PROGRAM pouStation2
VAR
	stationMode: FB_Mode;
	tCalcNumberOfPages: REAL;
	ceil: REAL;
	PartBuild: FB_PartBuild;
	retvall: UDINT;
	// TODO
	tPartPresent: BOOL;
	stationPower: FB_PowerDelay;
	
	task1: FB_Task;
	task2: FB_Task;
	task3: FB_Task;
	task4: FB_Task;
	task5: FB_Task;
	task6: FB_Task;
	task7: FB_Task;
	task8: FB_Task;
	task9: FB_Task;
	task10: FB_Task;
	task11: FB_Task;
	task12: FB_Task;
	task13: FB_Task;
	task14: FB_Task;
	task15: FB_Task;
	task16: FB_Task;
	task17: FB_Task;
	task18: FB_Task;
	task19: FB_Task;
	task20: FB_Task;
	checkTasks: FB_CheckTasks;
END_VAR

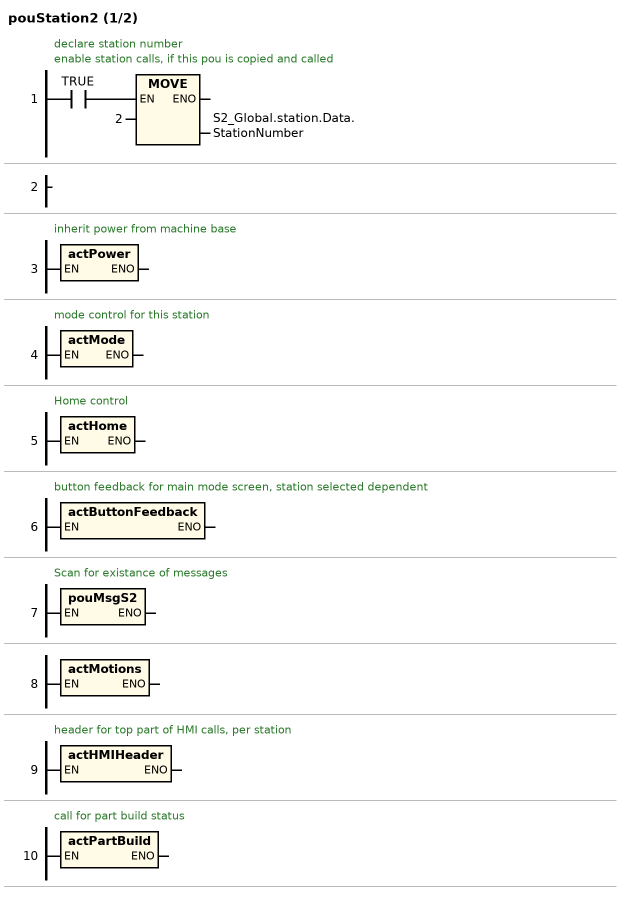
// NETWORK 1
// declare station number
// enable station calls, if this pou is copied and called
S2_Global.station.Data.StationNumber := 2;

// NETWORK 2

// NETWORK 3
// inherit power from machine base
actPower();

// NETWORK 4
// mode control for this station
actMode();

// NETWORK 5
// Home control
actHome();

// NETWORK 6
// button feedback for main mode screen, station selected dependent
actButtonFeedback();

// NETWORK 7
// Scan for existance of messages
pouMsgS2();

// NETWORK 8
actMotions();

// NETWORK 9
// header for top part of HMI calls, per station
actHMIHeader();

// NETWORK 10
// call for part build status
actPartBuild();

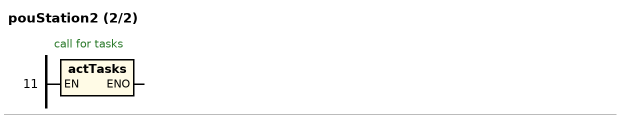
// NETWORK 11
// call for tasks
actTasks();

ACTION actButtonFeedback:
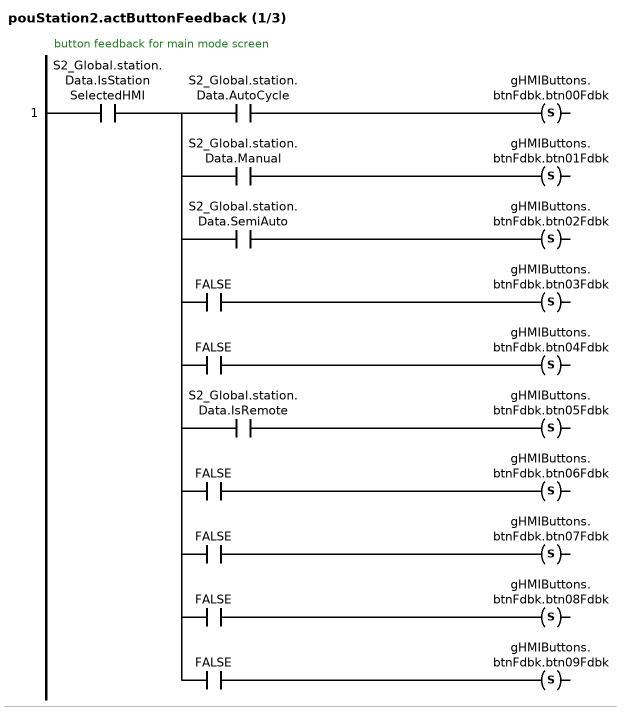
// NETWORK 1
// button feedback for main mode screen
gHMIButtons.btnFdbk.btn00Fdbk S= S2_Global.station.Data.IsStationSelectedHMI AND S2_Global.station.Data.AutoCycle;
gHMIButtons.btnFdbk.btn01Fdbk S= S2_Global.station.Data.IsStationSelectedHMI AND S2_Global.station.Data.Manual;
gHMIButtons.btnFdbk.btn02Fdbk S= S2_Global.station.Data.IsStationSelectedHMI AND S2_Global.station.Data.SemiAuto;
gHMIButtons.btnFdbk.btn03Fdbk S= S2_Global.station.Data.IsStationSelectedHMI AND FALSE;
gHMIButtons.btnFdbk.btn04Fdbk S= S2_Global.station.Data.IsStationSelectedHMI AND FALSE;
gHMIButtons.btnFdbk.btn05Fdbk S= S2_Global.station.Data.IsStationSelectedHMI AND S2_Global.station.Data.IsRemote;
gHMIButtons.btnFdbk.btn06Fdbk S= S2_Global.station.Data.IsStationSelectedHMI AND FALSE;
gHMIButtons.btnFdbk.btn07Fdbk S= S2_Global.station.Data.IsStationSelectedHMI AND FALSE;
gHMIButtons.btnFdbk.btn08Fdbk S= S2_Global.station.Data.IsStationSelectedHMI AND FALSE;
gHMIButtons.btnFdbk.btn09Fdbk S= S2_Global.station.Data.IsStationSelectedHMI AND FALSE;

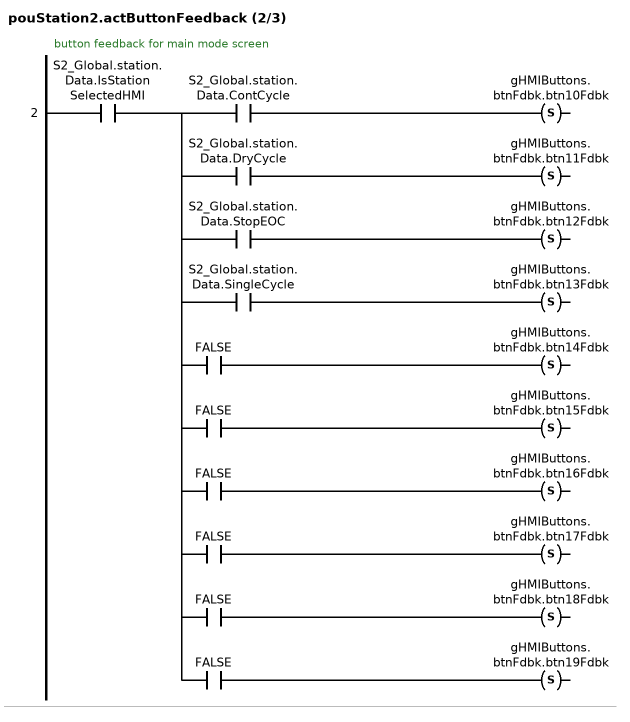
// NETWORK 2
// button feedback for main mode screen
gHMIButtons.btnFdbk.btn10Fdbk S= S2_Global.station.Data.IsStationSelectedHMI AND S2_Global.station.Data.ContCycle;
gHMIButtons.btnFdbk.btn11Fdbk S= S2_Global.station.Data.IsStationSelectedHMI AND S2_Global.station.Data.DryCycle;
gHMIButtons.btnFdbk.btn12Fdbk S= S2_Global.station.Data.IsStationSelectedHMI AND S2_Global.station.Data.StopEOC;
gHMIButtons.btnFdbk.btn13Fdbk S= S2_Global.station.Data.IsStationSelectedHMI AND S2_Global.station.Data.SingleCycle;
gHMIButtons.btnFdbk.btn14Fdbk S= S2_Global.station.Data.IsStationSelectedHMI AND FALSE;
gHMIButtons.btnFdbk.btn15Fdbk S= S2_Global.station.Data.IsStationSelectedHMI AND FALSE;
gHMIButtons.btnFdbk.btn16Fdbk S= S2_Global.station.Data.IsStationSelectedHMI AND FALSE;
gHMIButtons.btnFdbk.btn17Fdbk S= S2_Global.station.Data.IsStationSelectedHMI AND FALSE;
gHMIButtons.btnFdbk.btn18Fdbk S= S2_Global.station.Data.IsStationSelectedHMI AND FALSE;
gHMIButtons.btnFdbk.btn19Fdbk S= S2_Global.station.Data.IsStationSelectedHMI AND FALSE;

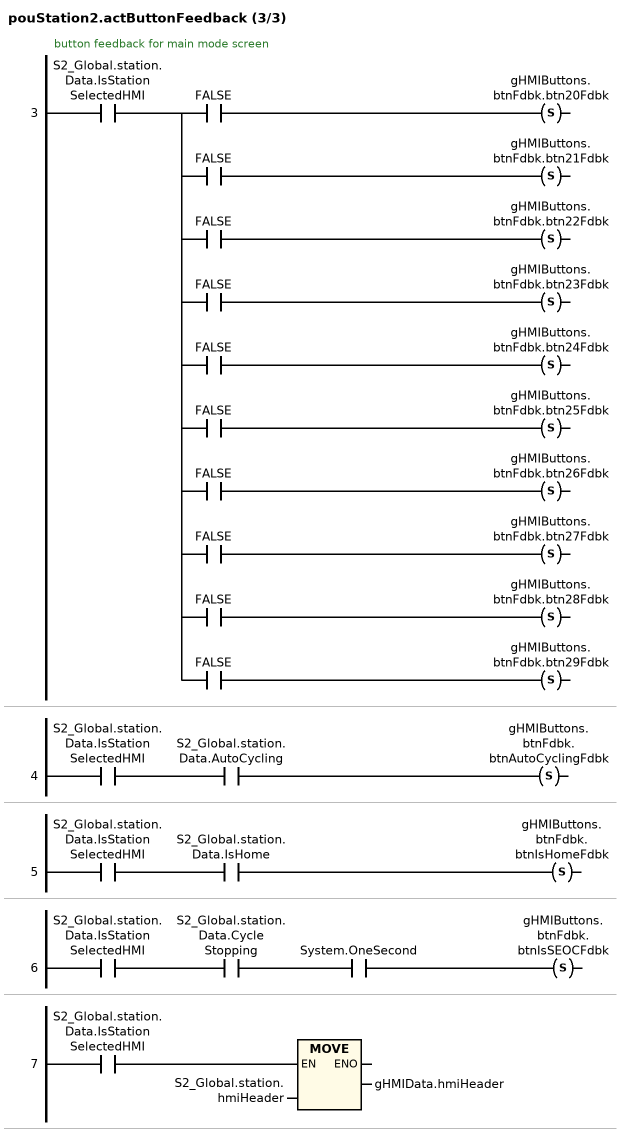
// NETWORK 3
// button feedback for main mode screen
gHMIButtons.btnFdbk.btn20Fdbk S= S2_Global.station.Data.IsStationSelectedHMI AND FALSE;
gHMIButtons.btnFdbk.btn21Fdbk S= S2_Global.station.Data.IsStationSelectedHMI AND FALSE;
gHMIButtons.btnFdbk.btn22Fdbk S= S2_Global.station.Data.IsStationSelectedHMI AND FALSE;
gHMIButtons.btnFdbk.btn23Fdbk S= S2_Global.station.Data.IsStationSelectedHMI AND FALSE;
gHMIButtons.btnFdbk.btn24Fdbk S= S2_Global.station.Data.IsStationSelectedHMI AND FALSE;
gHMIButtons.btnFdbk.btn25Fdbk S= S2_Global.station.Data.IsStationSelectedHMI AND FALSE;
gHMIButtons.btnFdbk.btn26Fdbk S= S2_Global.station.Data.IsStationSelectedHMI AND FALSE;
gHMIButtons.btnFdbk.btn27Fdbk S= S2_Global.station.Data.IsStationSelectedHMI AND FALSE;
gHMIButtons.btnFdbk.btn28Fdbk S= S2_Global.station.Data.IsStationSelectedHMI AND FALSE;
gHMIButtons.btnFdbk.btn29Fdbk S= S2_Global.station.Data.IsStationSelectedHMI AND FALSE;

// NETWORK 4
gHMIButtons.btnFdbk.btnAutoCyclingFdbk S= S2_Global.station.Data.IsStationSelectedHMI AND S2_Global.station.Data.AutoCycling;

// NETWORK 5
gHMIButtons.btnFdbk.btnIsHomeFdbk S= S2_Global.station.Data.IsStationSelectedHMI AND S2_Global.station.Data.IsHome;

// NETWORK 6
gHMIButtons.btnFdbk.btnIsSEOCFdbk S= S2_Global.station.Data.IsStationSelectedHMI AND S2_Global.station.Data.CycleStopping AND System.OneSecond;

// NETWORK 7
IF S2_Global.station.Data.IsStationSelectedHMI THEN gHMIData.hmiHeader := S2_Global.station.hmiHeader; END_IF
END_ACTION

ACTION actHMIHeader:
//set values on station
IF NOT S2_Global.station.Data.IsHome THEN
	S2_Global.station.hmiHeader.homestate := 0;
END_IF

IF S2_Global.station.Data.IsHoming THEN
	S2_Global.station.hmiHeader.homestate := 1;
END_IF

IF S2_Global.station.Data.IsHome THEN
	S2_Global.station.hmiHeader.homestate := 2;
END_IF

IF	S2_Global.station.Data.IsHome OR
	S2_Global.station.Data.IsHoming AND System.OneSecond THEN
	S2_Global.station.hmiHeader.homestateColour := TRUE;
	ELSE
	S2_Global.station.hmiHeader.homestateColour := FALSE;	
END_IF

IF S2_Global.station.Data.Fault THEN
	S2_Global.station.hmiHeader.FaultStateHeader := 1;
	ELSE
	S2_Global.station.hmiHeader.FaultStateHeader := 0;
END_IF

IF S2_Global.station.Data.Fault THEN
	S2_Global.station.hmiHeader.isFaultState := TRUE;
	ELSE
	S2_Global.station.hmiHeader.isFaultState := FALSE;
END_IF

IF	S2_Global.station.Data.CycleStopping AND System.OneSecond THEN
	S2_Global.station.hmiHeader.stationstateColour := TRUE;
	ELSE
	S2_Global.station.hmiHeader.stationstateColour := FALSE;	
END_IF


S2_Global.station.hmiHeader.stationNameSelect := S2_Global.station.Data.StationNumber;
S2_Global.station.hmiHeader.stationstate := S2_Global.station.Data.StationState;

S2_Global.station.hmiHeader.flasher := System.OneSecond;
END_ACTION

ACTION actHome:
//Set home status for station

IF 
//are all motions returned
S2_01_Motion_1.Motion.qReturnDepth AND
S2_01_Motion_2.Motion.qReturnDepth AND
S2_01_Motion_3.Motion.qReturnDepth AND
S2_01_Motion_4.Motion.qReturnDepth AND
S2_01_Motion_5.Motion.qReturnDepth AND
S2_01_Motion_6.Motion.qReturnDepth

	THEN
		//set IsHome value for station
		S2_Global.station.Data.IsHome := TRUE;
	ELSE
		S2_Global.station.Data.IsHome := FALSE;
END_IF
END_ACTION

ACTION actMaxNumStationPages:
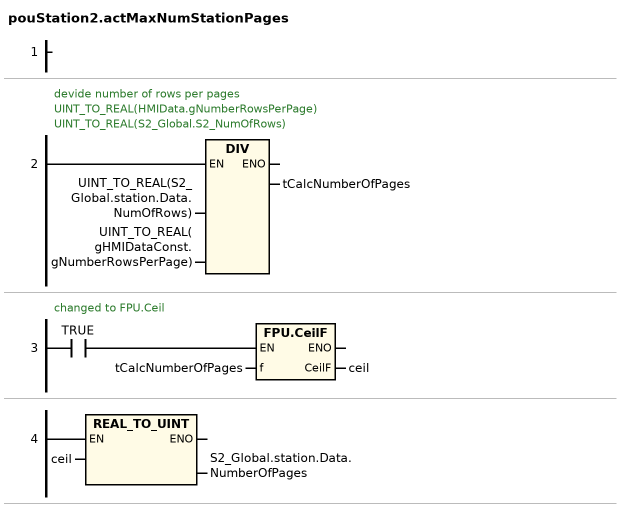
// NETWORK 1

// NETWORK 2
// devide number of rows per pages
// UINT_TO_REAL(HMIData.gNumberRowsPerPage)
// UINT_TO_REAL(S2_Global.S2_NumOfRows)
tCalcNumberOfPages := (UINT_TO_REAL(S2_Global.station.Data.NumOfRows)) / (UINT_TO_REAL(gHMIDataConst.gNumberRowsPerPage));

// NETWORK 3
// changed to FPU.Ceil
ceil := FPU.CeilF(f := tCalcNumberOfPages);

// NETWORK 4
S2_Global.station.Data.NumberOfPages := REAL_TO_UINT(ceil);
END_ACTION

ACTION actMode:
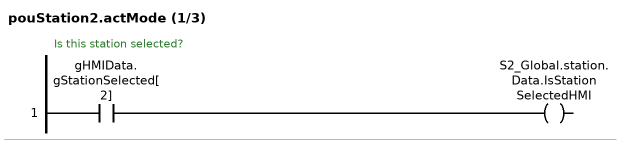
// NETWORK 1
// Is this station selected?
S2_Global.station.Data.IsStationSelectedHMI := gHMIData.gStationSelected[2];

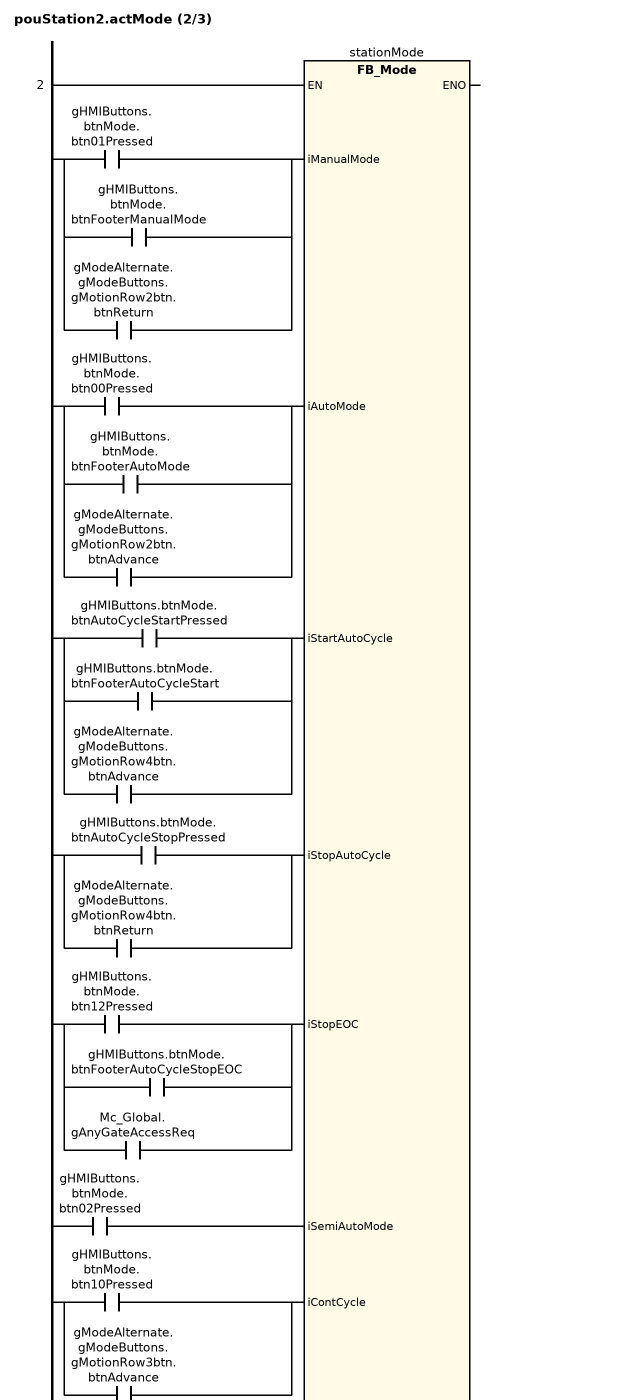
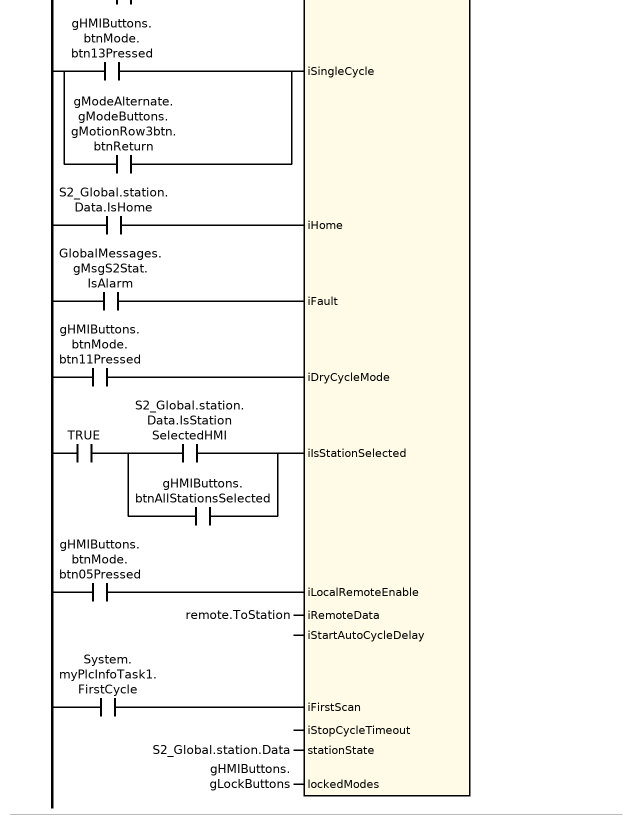
// NETWORK 2
stationMode(
    iManualMode := gHMIButtons.btnMode.btn01Pressed OR gHMIButtons.btnMode.btnFooterManualMode OR gModeAlternate.gModeButtons.gMotionRow2btn.btnReturn,
    iAutoMode := gHMIButtons.btnMode.btn00Pressed OR gHMIButtons.btnMode.btnFooterAutoMode OR gModeAlternate.gModeButtons.gMotionRow2btn.btnAdvance,
    iStartAutoCycle := gHMIButtons.btnMode.btnAutoCycleStartPressed OR gHMIButtons.btnMode.btnFooterAutoCycleStart OR gModeAlternate.gModeButtons.gMotionRow4btn.btnAdvance,
    iStopAutoCycle := gHMIButtons.btnMode.btnAutoCycleStopPressed OR gModeAlternate.gModeButtons.gMotionRow4btn.btnReturn,
    iStopEOC := gHMIButtons.btnMode.btn12Pressed OR gHMIButtons.btnMode.btnFooterAutoCycleStopEOC OR Mc_Global.gAnyGateAccessReq,
    iSemiAutoMode := gHMIButtons.btnMode.btn02Pressed,
    iContCycle := gHMIButtons.btnMode.btn10Pressed OR gModeAlternate.gModeButtons.gMotionRow3btn.btnAdvance,
    iSingleCycle := gHMIButtons.btnMode.btn13Pressed OR gModeAlternate.gModeButtons.gMotionRow3btn.btnReturn,
    iHome := S2_Global.station.Data.IsHome,
    iFault := GlobalMessages.gMsgS2Stat.IsAlarm,
    iDryCycleMode := gHMIButtons.btnMode.btn11Pressed,
    iIsStationSelected := TRUE AND (S2_Global.station.Data.IsStationSelectedHMI OR gHMIButtons.btnAllStationsSelected),
    iLocalRemoteEnable := gHMIButtons.btnMode.btn05Pressed,
    iRemoteData := remote.ToStation,
    iFirstScan := System.myPlcInfoTask1.FirstCycle,
    stationState := S2_Global.station.Data,
    lockedModes := gHMIButtons.gLockButtons); // FB_Mode

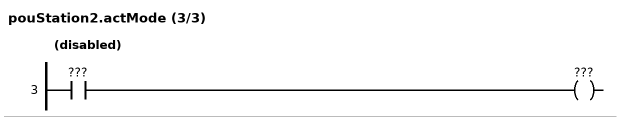
// NETWORK 3 (disabled)
// ??? := ???;
END_ACTION

ACTION actMotions:
//station 2 = 20000 index

//init number of rows
S2_Global.station.Data.NumOfRows := 0;

//set to 0
S2_global.station.dynRowNumber := 0;

//page 1
IF System.gSetup.stationFunctions[2].numRowsConfig >= 1 THEN S2_01_Motion_1(); END_IF
IF System.gSetup.stationFunctions[2].numRowsConfig >= 2 THEN S2_01_Motion_2(); END_IF
IF System.gSetup.stationFunctions[2].numRowsConfig >= 3 THEN S2_01_Motion_3(); END_IF
IF System.gSetup.stationFunctions[2].numRowsConfig >= 4 THEN S2_01_Motion_4(); END_IF
IF System.gSetup.stationFunctions[2].numRowsConfig >= 5 THEN S2_01_Motion_5(); END_IF
IF System.gSetup.stationFunctions[2].numRowsConfig >= 6 THEN S2_01_Motion_6(); END_IF
IF System.gSetup.stationFunctions[2].numRowsConfig >= 7 THEN S2_01_Motion_7(); END_IF
IF System.gSetup.stationFunctions[2].numRowsConfig >= 8 THEN S2_01_Motion_8(); END_IF
IF System.gSetup.stationFunctions[2].numRowsConfig >= 9 THEN S2_01_Motion_9(); END_IF

//page 2
IF System.gSetup.stationFunctions[2].numRowsConfig >= 10 THEN S2_01_Motion_10(); END_IF
IF System.gSetup.stationFunctions[2].numRowsConfig >= 11 THEN S2_01_Motion_11(); END_IF
IF System.gSetup.stationFunctions[2].numRowsConfig >= 12 THEN S2_01_Motion_12(); END_IF
IF System.gSetup.stationFunctions[2].numRowsConfig >= 13 THEN S2_01_Motion_13(); END_IF
IF System.gSetup.stationFunctions[2].numRowsConfig >= 14 THEN S2_01_Motion_14(); END_IF
IF System.gSetup.stationFunctions[2].numRowsConfig >= 15 THEN S2_01_Motion_15(); END_IF
IF System.gSetup.stationFunctions[2].numRowsConfig >= 16 THEN S2_01_Motion_16(); END_IF
IF System.gSetup.stationFunctions[2].numRowsConfig >= 17 THEN S2_01_Motion_17(); END_IF
IF System.gSetup.stationFunctions[2].numRowsConfig >= 18 THEN S2_01_Motion_18(); END_IF
IF System.gSetup.stationFunctions[2].numRowsConfig >= 19 THEN S2_01_Motion_19(); END_IF

//page 3
IF System.gSetup.stationFunctions[2].numRowsConfig >= 20 THEN S2_01_Motion_20(); END_IF
IF System.gSetup.stationFunctions[2].numRowsConfig >= 21 THEN S2_01_Motion_21(); END_IF
IF System.gSetup.stationFunctions[2].numRowsConfig >= 22 THEN S2_01_Motion_22(); END_IF
IF System.gSetup.stationFunctions[2].numRowsConfig >= 23 THEN S2_01_Motion_23(); END_IF
IF System.gSetup.stationFunctions[2].numRowsConfig >= 24 THEN S2_01_Motion_24(); END_IF
IF System.gSetup.stationFunctions[2].numRowsConfig >= 25 THEN S2_01_Motion_25(); END_IF
IF System.gSetup.stationFunctions[2].numRowsConfig >= 26 THEN S2_01_Motion_26(); END_IF
IF System.gSetup.stationFunctions[2].numRowsConfig >= 27 THEN S2_01_Motion_27(); END_IF
IF System.gSetup.stationFunctions[2].numRowsConfig >= 28 THEN S2_01_Motion_28(); END_IF
IF System.gSetup.stationFunctions[2].numRowsConfig >= 29 THEN S2_01_Motion_29(); END_IF

//page 4
IF System.gSetup.stationFunctions[2].numRowsConfig >= 30 THEN S2_01_Motion_30(); END_IF
IF System.gSetup.stationFunctions[2].numRowsConfig >= 31 THEN S2_01_Motion_31(); END_IF
IF System.gSetup.stationFunctions[2].numRowsConfig >= 32 THEN S2_01_Motion_32(); END_IF
IF System.gSetup.stationFunctions[2].numRowsConfig >= 33 THEN S2_01_Motion_33(); END_IF
IF System.gSetup.stationFunctions[2].numRowsConfig >= 34 THEN S2_01_Motion_34(); END_IF
IF System.gSetup.stationFunctions[2].numRowsConfig >= 35 THEN S2_01_Motion_35(); END_IF
IF System.gSetup.stationFunctions[2].numRowsConfig >= 36 THEN S2_01_Motion_36(); END_IF
IF System.gSetup.stationFunctions[2].numRowsConfig >= 37 THEN S2_01_Motion_37(); END_IF
IF System.gSetup.stationFunctions[2].numRowsConfig >= 38 THEN S2_01_Motion_38(); END_IF
IF System.gSetup.stationFunctions[2].numRowsConfig >= 39 THEN S2_01_Motion_39(); END_IF

//page 5
IF System.gSetup.stationFunctions[2].numRowsConfig >= 40 THEN S2_01_Motion_40(); END_IF
IF System.gSetup.stationFunctions[2].numRowsConfig >= 41 THEN S2_01_Motion_41(); END_IF
IF System.gSetup.stationFunctions[2].numRowsConfig >= 42 THEN S2_01_Motion_42(); END_IF
IF System.gSetup.stationFunctions[2].numRowsConfig >= 43 THEN S2_01_Motion_43(); END_IF
IF System.gSetup.stationFunctions[2].numRowsConfig >= 44 THEN S2_01_Motion_44(); END_IF
IF System.gSetup.stationFunctions[2].numRowsConfig >= 45 THEN S2_01_Motion_45(); END_IF
IF System.gSetup.stationFunctions[2].numRowsConfig >= 46 THEN S2_01_Motion_46(); END_IF
IF System.gSetup.stationFunctions[2].numRowsConfig >= 47 THEN S2_01_Motion_47(); END_IF
IF System.gSetup.stationFunctions[2].numRowsConfig >= 48 THEN S2_01_Motion_48(); END_IF
IF System.gSetup.stationFunctions[2].numRowsConfig >= 49 THEN S2_01_Motion_49(); END_IF

//page 6
IF System.gSetup.stationFunctions[2].numRowsConfig >= 50 THEN S2_01_Motion_50(); END_IF
IF System.gSetup.stationFunctions[2].numRowsConfig >= 51 THEN S2_01_Motion_51(); END_IF
IF System.gSetup.stationFunctions[2].numRowsConfig >= 52 THEN S2_01_Motion_52(); END_IF
IF System.gSetup.stationFunctions[2].numRowsConfig >= 53 THEN S2_01_Motion_53(); END_IF
IF System.gSetup.stationFunctions[2].numRowsConfig >= 54 THEN S2_01_Motion_54(); END_IF
IF System.gSetup.stationFunctions[2].numRowsConfig >= 55 THEN S2_01_Motion_55(); END_IF
IF System.gSetup.stationFunctions[2].numRowsConfig >= 56 THEN S2_01_Motion_56(); END_IF
IF System.gSetup.stationFunctions[2].numRowsConfig >= 57 THEN S2_01_Motion_57(); END_IF
IF System.gSetup.stationFunctions[2].numRowsConfig >= 58 THEN S2_01_Motion_58(); END_IF
IF System.gSetup.stationFunctions[2].numRowsConfig >= 59 THEN S2_01_Motion_59(); END_IF

//page 7
IF System.gSetup.stationFunctions[2].numRowsConfig >= 60 THEN S2_01_Motion_60(); END_IF
IF System.gSetup.stationFunctions[2].numRowsConfig >= 61 THEN S2_01_Motion_61(); END_IF
IF System.gSetup.stationFunctions[2].numRowsConfig >= 62 THEN S2_01_Motion_62(); END_IF
IF System.gSetup.stationFunctions[2].numRowsConfig >= 63 THEN S2_01_Motion_63(); END_IF
IF System.gSetup.stationFunctions[2].numRowsConfig >= 64 THEN S2_01_Motion_64(); END_IF
IF System.gSetup.stationFunctions[2].numRowsConfig >= 65 THEN S2_01_Motion_65(); END_IF
IF System.gSetup.stationFunctions[2].numRowsConfig >= 66 THEN S2_01_Motion_66(); END_IF
IF System.gSetup.stationFunctions[2].numRowsConfig >= 67 THEN S2_01_Motion_67(); END_IF
IF System.gSetup.stationFunctions[2].numRowsConfig >= 68 THEN S2_01_Motion_68(); END_IF
IF System.gSetup.stationFunctions[2].numRowsConfig >= 69 THEN S2_01_Motion_69(); END_IF

//page 8
IF System.gSetup.stationFunctions[2].numRowsConfig >= 70 THEN S2_01_Motion_70(); END_IF
IF System.gSetup.stationFunctions[2].numRowsConfig >= 71 THEN S2_01_Motion_71(); END_IF
IF System.gSetup.stationFunctions[2].numRowsConfig >= 72 THEN S2_01_Motion_72(); END_IF
IF System.gSetup.stationFunctions[2].numRowsConfig >= 73 THEN S2_01_Motion_73(); END_IF
IF System.gSetup.stationFunctions[2].numRowsConfig >= 74 THEN S2_01_Motion_74(); END_IF
IF System.gSetup.stationFunctions[2].numRowsConfig >= 75 THEN S2_01_Motion_75(); END_IF
IF System.gSetup.stationFunctions[2].numRowsConfig >= 76 THEN S2_01_Motion_76(); END_IF
IF System.gSetup.stationFunctions[2].numRowsConfig >= 77 THEN S2_01_Motion_77(); END_IF
IF System.gSetup.stationFunctions[2].numRowsConfig >= 78 THEN S2_01_Motion_78(); END_IF
IF System.gSetup.stationFunctions[2].numRowsConfig >= 79 THEN S2_01_Motion_79(); END_IF

//page 9
IF System.gSetup.stationFunctions[2].numRowsConfig >= 80 THEN S2_01_Motion_80(); END_IF
IF System.gSetup.stationFunctions[2].numRowsConfig >= 81 THEN S2_01_Motion_81(); END_IF
IF System.gSetup.stationFunctions[2].numRowsConfig >= 82 THEN S2_01_Motion_82(); END_IF
IF System.gSetup.stationFunctions[2].numRowsConfig >= 83 THEN S2_01_Motion_83(); END_IF
IF System.gSetup.stationFunctions[2].numRowsConfig >= 84 THEN S2_01_Motion_84(); END_IF
IF System.gSetup.stationFunctions[2].numRowsConfig >= 85 THEN S2_01_Motion_85(); END_IF
IF System.gSetup.stationFunctions[2].numRowsConfig >= 86 THEN S2_01_Motion_86(); END_IF
IF System.gSetup.stationFunctions[2].numRowsConfig >= 87 THEN S2_01_Motion_87(); END_IF
IF System.gSetup.stationFunctions[2].numRowsConfig >= 88 THEN S2_01_Motion_88(); END_IF
IF System.gSetup.stationFunctions[2].numRowsConfig >= 89 THEN S2_01_Motion_89(); END_IF

//page 10
IF System.gSetup.stationFunctions[2].numRowsConfig >= 90 THEN S2_01_Motion_90(); END_IF
IF System.gSetup.stationFunctions[2].numRowsConfig >= 91 THEN S2_01_Motion_91(); END_IF
IF System.gSetup.stationFunctions[2].numRowsConfig >= 92 THEN S2_01_Motion_92(); END_IF
IF System.gSetup.stationFunctions[2].numRowsConfig >= 93 THEN S2_01_Motion_93(); END_IF
IF System.gSetup.stationFunctions[2].numRowsConfig >= 94 THEN S2_01_Motion_94(); END_IF
IF System.gSetup.stationFunctions[2].numRowsConfig >= 95 THEN S2_01_Motion_95(); END_IF
IF System.gSetup.stationFunctions[2].numRowsConfig >= 96 THEN S2_01_Motion_96(); END_IF
IF System.gSetup.stationFunctions[2].numRowsConfig >= 97 THEN S2_01_Motion_97(); END_IF
IF System.gSetup.stationFunctions[2].numRowsConfig >= 98 THEN S2_01_Motion_98(); END_IF
IF System.gSetup.stationFunctions[2].numRowsConfig >= 99 THEN S2_01_Motion_99(); END_IF

//must be called after motionRow calls
actMaxNumStationPages();
END_ACTION

ACTION actPartBuild:
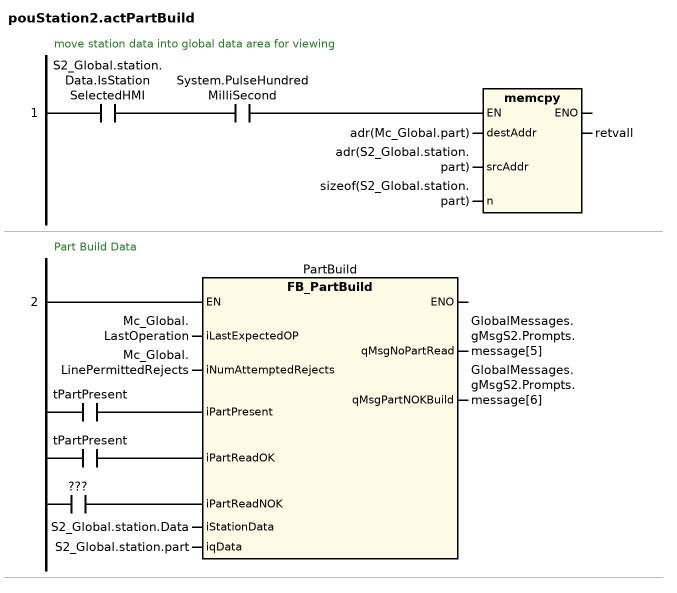
// NETWORK 1
// move station data into global data area for viewing
IF S2_Global.station.Data.IsStationSelectedHMI AND System.PulseHundredMilliSecond THEN
    retvall := memcpy(destAddr := adr(Mc_Global.part), srcAddr := adr(S2_Global.station.part), n := sizeof(S2_Global.station.part));
END_IF

// NETWORK 2
// Part Build Data
PartBuild(
    iLastExpectedOP := Mc_Global.LastOperation,
    iNumAttemptedRejects := Mc_Global.LinePermittedRejects,
    iPartPresent := tPartPresent,
    iPartReadOK := tPartPresent,
    iStationData := S2_Global.station.Data,
    iqData := S2_Global.station.part,
    qMsgNoPartRead => GlobalMessages.gMsgS2.Prompts.message[5],
    qMsgPartNOKBuild => GlobalMessages.gMsgS2.Prompts.message[6]); // FB_PartBuild
END_ACTION

ACTION actPower:
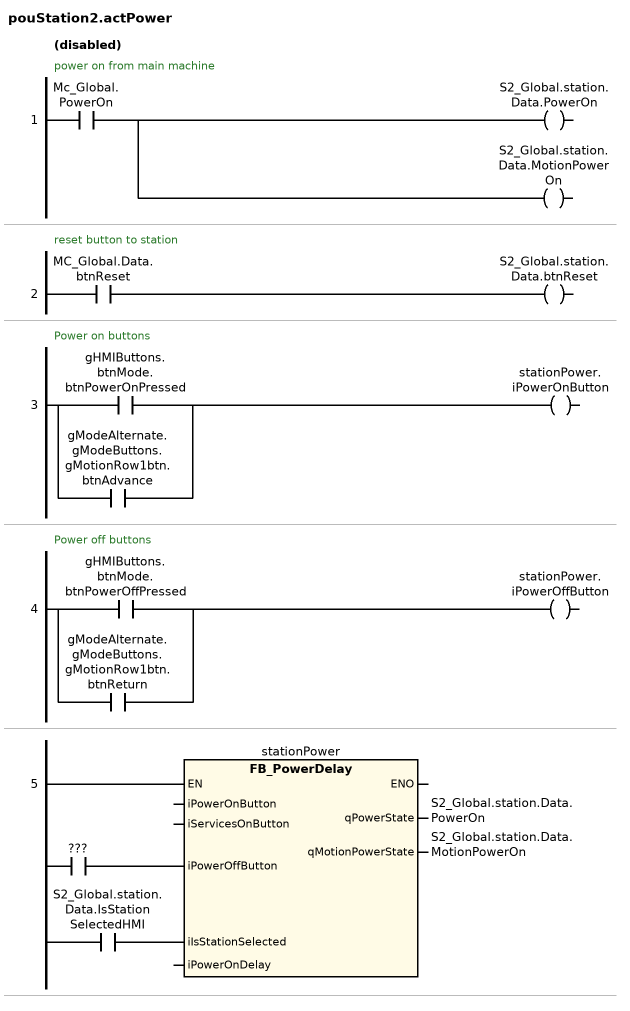
// NETWORK 1 (disabled)
// power on from main machine
// S2_Global.station.Data.PowerOn := Mc_Global.PowerOn;
// S2_Global.station.Data.MotionPowerOn := Mc_Global.PowerOn;

// NETWORK 2
// reset button to station
S2_Global.station.Data.btnReset := MC_Global.Data.btnReset;

// NETWORK 3
// Power on buttons
stationPower.iPowerOnButton := gHMIButtons.btnMode.btnPowerOnPressed OR gModeAlternate.gModeButtons.gMotionRow1btn.btnAdvance;

// NETWORK 4
// Power off buttons
stationPower.iPowerOffButton := gHMIButtons.btnMode.btnPowerOffPressed OR gModeAlternate.gModeButtons.gMotionRow1btn.btnReturn;

// NETWORK 5
stationPower(
    iIsStationSelected := S2_Global.station.Data.IsStationSelectedHMI,
    qPowerState => S2_Global.station.Data.PowerOn,
    qMotionPowerState => S2_Global.station.Data.MotionPowerOn); // FB_PowerDelay
END_ACTION

ACTION actTasks:
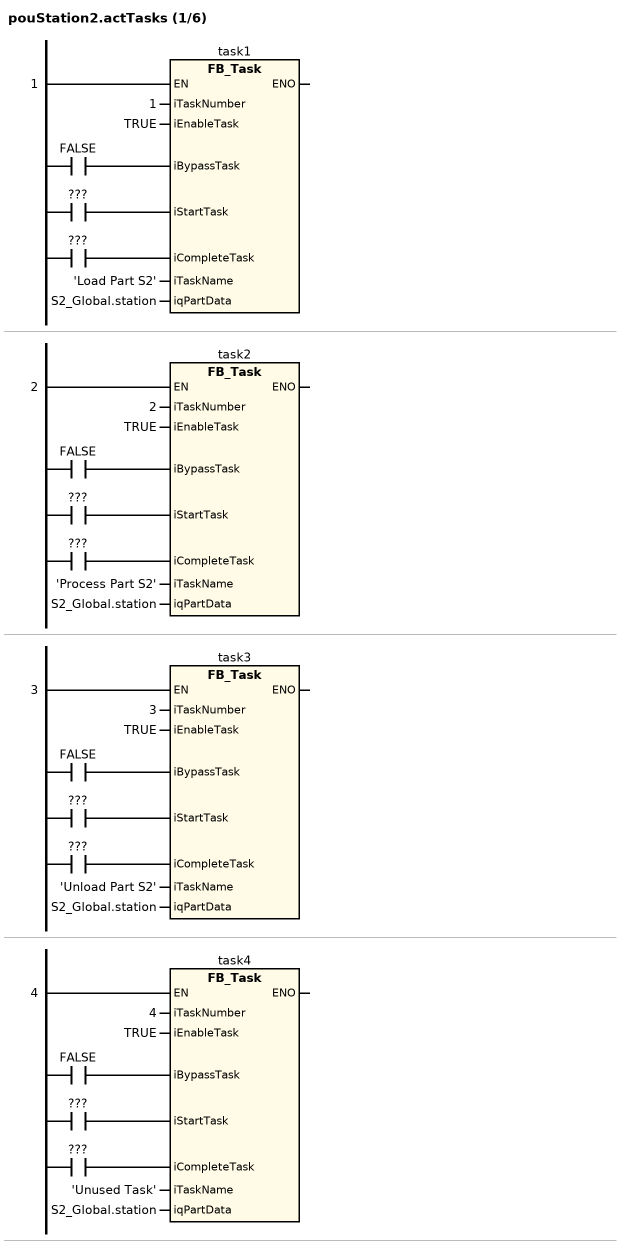
// NETWORK 1
task1(
    iTaskNumber := 1,
    iEnableTask := TRUE,
    iBypassTask := FALSE,
    iTaskName := 'Load Part S2',
    iqPartData := S2_Global.station); // FB_Task

// NETWORK 2
task2(
    iTaskNumber := 2,
    iEnableTask := TRUE,
    iBypassTask := FALSE,
    iTaskName := 'Process Part S2',
    iqPartData := S2_Global.station); // FB_Task

// NETWORK 3
task3(
    iTaskNumber := 3,
    iEnableTask := TRUE,
    iBypassTask := FALSE,
    iTaskName := 'Unload Part S2',
    iqPartData := S2_Global.station); // FB_Task

// NETWORK 4
task4(
    iTaskNumber := 4,
    iEnableTask := TRUE,
    iBypassTask := FALSE,
    iTaskName := 'Unused Task',
    iqPartData := S2_Global.station); // FB_Task

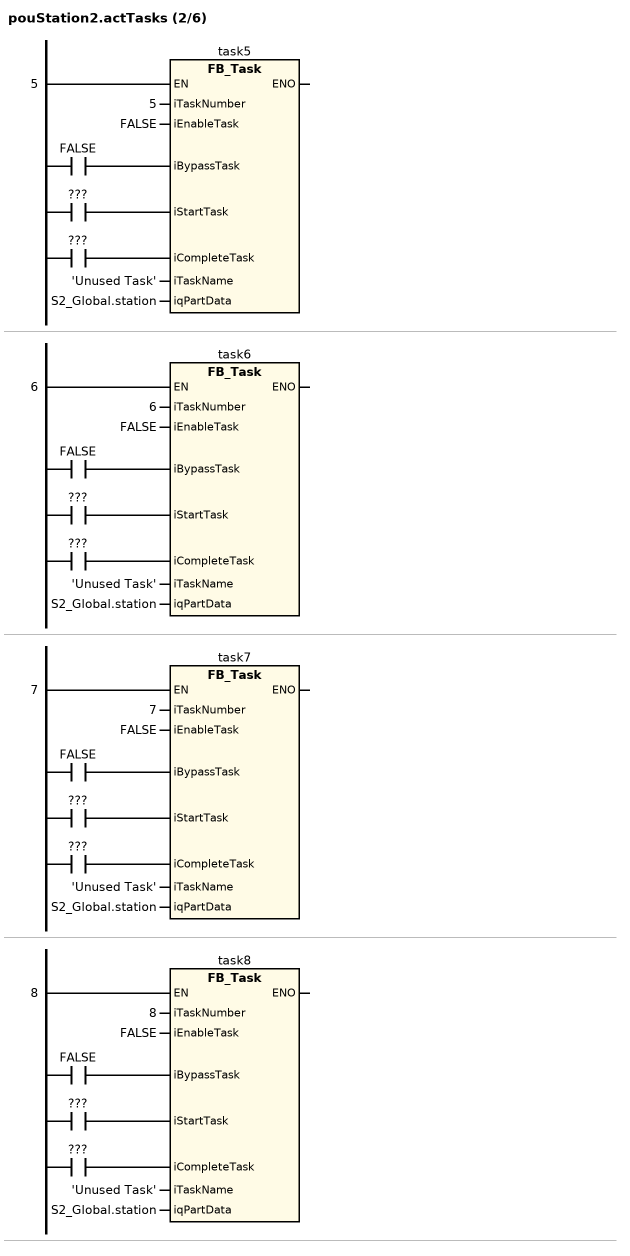
// NETWORK 5
task5(
    iTaskNumber := 5,
    iEnableTask := FALSE,
    iBypassTask := FALSE,
    iTaskName := 'Unused Task',
    iqPartData := S2_Global.station); // FB_Task

// NETWORK 6
task6(
    iTaskNumber := 6,
    iEnableTask := FALSE,
    iBypassTask := FALSE,
    iTaskName := 'Unused Task',
    iqPartData := S2_Global.station); // FB_Task

// NETWORK 7
task7(
    iTaskNumber := 7,
    iEnableTask := FALSE,
    iBypassTask := FALSE,
    iTaskName := 'Unused Task',
    iqPartData := S2_Global.station); // FB_Task

// NETWORK 8
task8(
    iTaskNumber := 8,
    iEnableTask := FALSE,
    iBypassTask := FALSE,
    iTaskName := 'Unused Task',
    iqPartData := S2_Global.station); // FB_Task

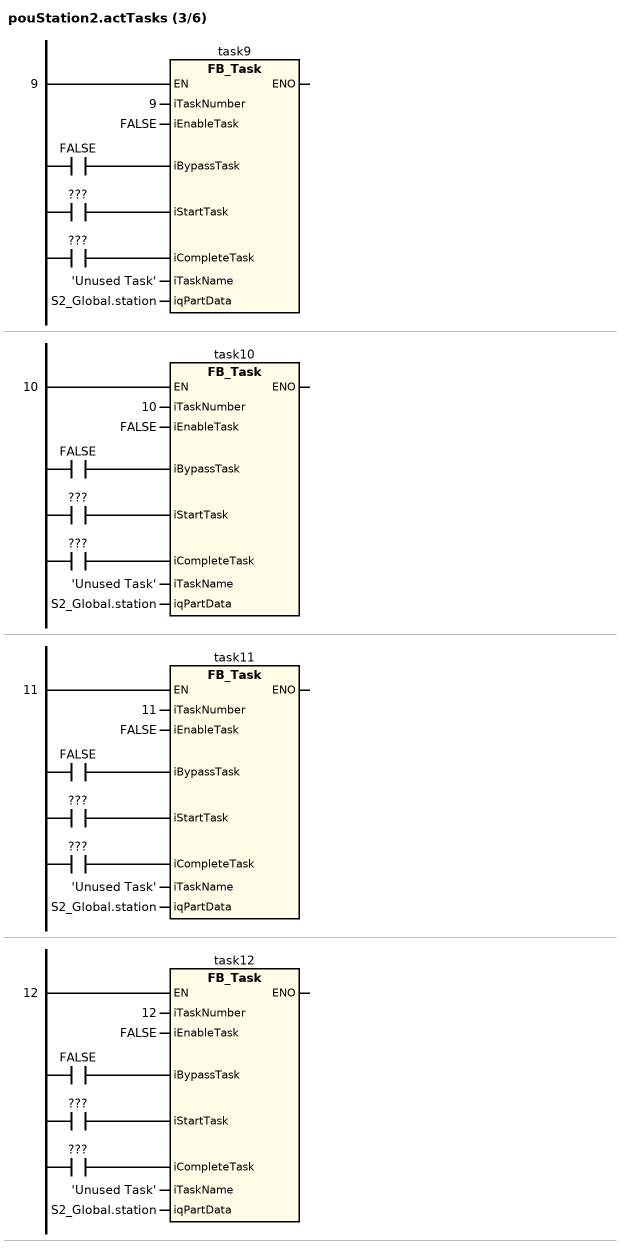
// NETWORK 9
task9(
    iTaskNumber := 9,
    iEnableTask := FALSE,
    iBypassTask := FALSE,
    iTaskName := 'Unused Task',
    iqPartData := S2_Global.station); // FB_Task

// NETWORK 10
task10(
    iTaskNumber := 10,
    iEnableTask := FALSE,
    iBypassTask := FALSE,
    iTaskName := 'Unused Task',
    iqPartData := S2_Global.station); // FB_Task

// NETWORK 11
task11(
    iTaskNumber := 11,
    iEnableTask := FALSE,
    iBypassTask := FALSE,
    iTaskName := 'Unused Task',
    iqPartData := S2_Global.station); // FB_Task

// NETWORK 12
task12(
    iTaskNumber := 12,
    iEnableTask := FALSE,
    iBypassTask := FALSE,
    iTaskName := 'Unused Task',
    iqPartData := S2_Global.station); // FB_Task

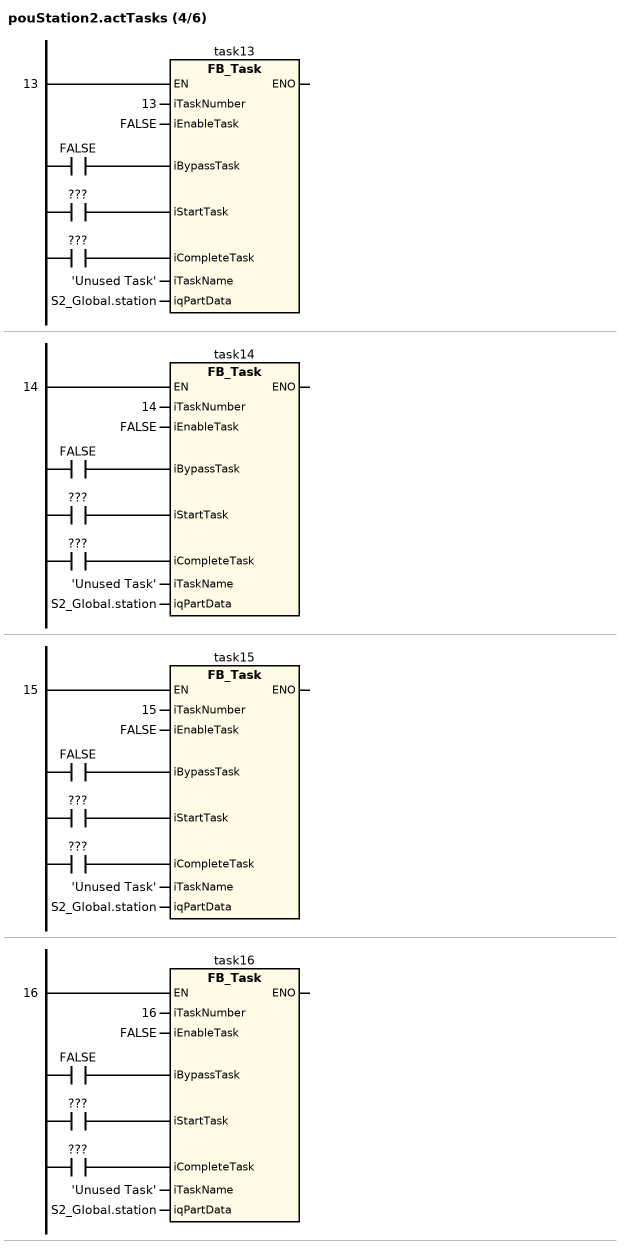
// NETWORK 13
task13(
    iTaskNumber := 13,
    iEnableTask := FALSE,
    iBypassTask := FALSE,
    iTaskName := 'Unused Task',
    iqPartData := S2_Global.station); // FB_Task

// NETWORK 14
task14(
    iTaskNumber := 14,
    iEnableTask := FALSE,
    iBypassTask := FALSE,
    iTaskName := 'Unused Task',
    iqPartData := S2_Global.station); // FB_Task

// NETWORK 15
task15(
    iTaskNumber := 15,
    iEnableTask := FALSE,
    iBypassTask := FALSE,
    iTaskName := 'Unused Task',
    iqPartData := S2_Global.station); // FB_Task

// NETWORK 16
task16(
    iTaskNumber := 16,
    iEnableTask := FALSE,
    iBypassTask := FALSE,
    iTaskName := 'Unused Task',
    iqPartData := S2_Global.station); // FB_Task

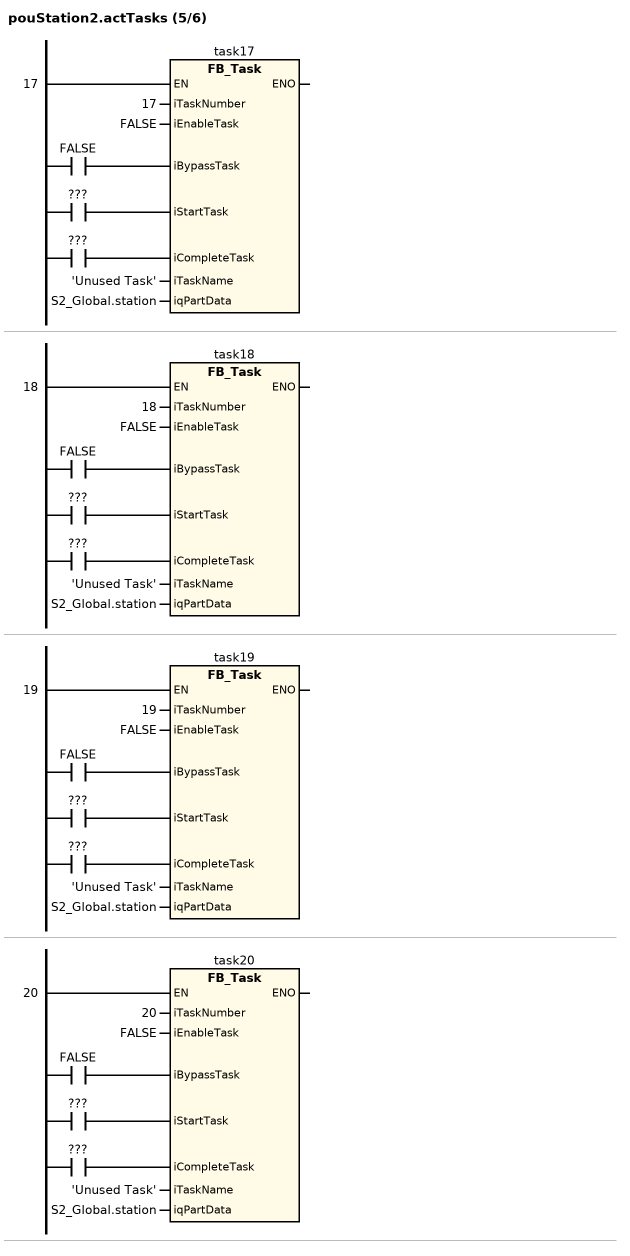
// NETWORK 17
task17(
    iTaskNumber := 17,
    iEnableTask := FALSE,
    iBypassTask := FALSE,
    iTaskName := 'Unused Task',
    iqPartData := S2_Global.station); // FB_Task

// NETWORK 18
task18(
    iTaskNumber := 18,
    iEnableTask := FALSE,
    iBypassTask := FALSE,
    iTaskName := 'Unused Task',
    iqPartData := S2_Global.station); // FB_Task

// NETWORK 19
task19(
    iTaskNumber := 19,
    iEnableTask := FALSE,
    iBypassTask := FALSE,
    iTaskName := 'Unused Task',
    iqPartData := S2_Global.station); // FB_Task

// NETWORK 20
task20(
    iTaskNumber := 20,
    iEnableTask := FALSE,
    iBypassTask := FALSE,
    iTaskName := 'Unused Task',
    iqPartData := S2_Global.station); // FB_Task

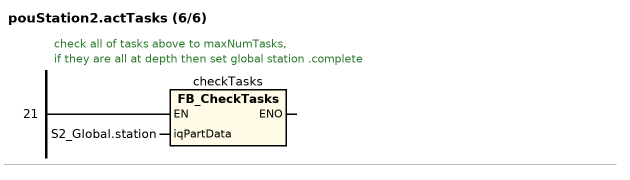
// NETWORK 21
// check all of tasks above to maxNumTasks,
// if they are all at depth then set global station .complete
checkTasks(iqPartData := S2_Global.station); // FB_CheckTasks
END_ACTION

END_PROGRAM

(* stored: Version 1.1.0.1, ProductVersion 3.1.4024.11
   POU pouStation2: Id {fd8ca611-dcd7-4808-b220-3ca7fa511e9d}, SpecialFunc None
   Action actButtonFeedback: Id {53e81109-c13a-4493-b591-48fbf4002db6}
   Action actHMIHeader: Id {2f2a041f-294e-40ca-9801-641257a802ed}
   Action actHome: Id {0883900f-8058-40f6-a4c3-fae5254b2ba8}
   Action actMaxNumStationPages: Id {7ce2426d-b6e4-45d9-acfd-953f5fdcae61}
   Action actMode: Id {89491c54-f09e-4480-a81d-ba1f3bfa5019}
   Action actMotions: Id {66fa6756-b646-460a-b835-0014fc22e25b}
   Action actPartBuild: Id {f0f8c37e-cd13-490d-a003-cb5f08cd140b}
   Action actPower: Id {7bbc8cd9-3e8d-40ea-83fb-9a607850df83}
   Action actTasks: Id {1f5ba35b-7118-4969-8414-8b916b3b8aa7} *)
